(* PLC project Sem nome, Desconhecido Sem nome 1 *)
(* stored: creationDateTime 2019-06-13T18:39:07, modificationDateTime 2019-06-23T17:14:26 *)

PROGRAM program0
  VAR
    saida AT %QX100.0 : BOOL;
    setpoint AT %QW4 : UINT;
    Temperatura AT %IW100 : UINT;
    SaidaAnalog AT %QW100 : UINT;
    Erro AT %QW20 : INT;
    saida2 AT %QX101.0 : BOOL;
    setpoint2 AT %QW8 : UINT;
    Temperatura2 AT %IW102 : UINT;
    SaidaAnalog2 AT %QW101 : UINT;
    Erro2 AT %QW30 : INT;
    aux1 AT %MW200 : UINT;
    aux2 AT %MX202.0 : BOOL;
    aux3 AT %MW204 : UINT;
    aux4 AT %MX202.1 : BOOL;
  END_VAR

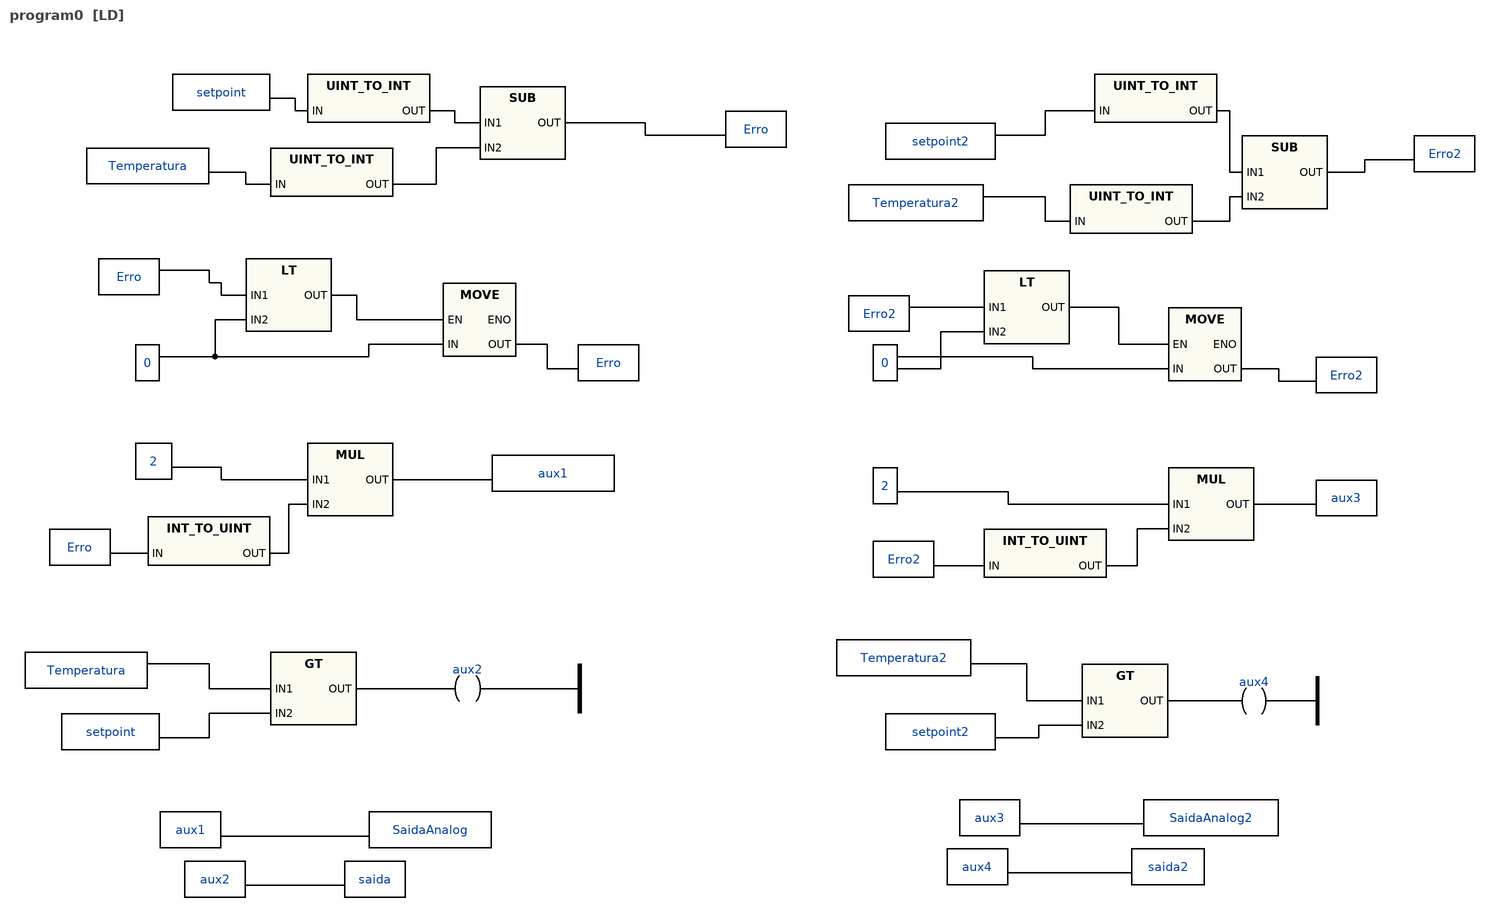
(* LD diagram, written out as Structured Text *)
Erro := UINT_TO_INT(setpoint) - UINT_TO_INT(Temperatura);
Erro2 := UINT_TO_INT(setpoint2) - UINT_TO_INT(Temperatura2);
IF Erro < 0 THEN Erro := 0; END_IF;
IF Erro2 < 0 THEN Erro2 := 0; END_IF;
aux1 := 2 * INT_TO_UINT(Erro);
aux3 := 2 * INT_TO_UINT(Erro2);
aux2 := Temperatura > setpoint;
aux4 := Temperatura2 > setpoint2;
SaidaAnalog2 := aux3;
SaidaAnalog := aux1;
saida2 := aux4;
saida := aux2;
END_PROGRAM

CONFIGURATION Config0
  RESOURCE Res0 ON PLC
    TASK task0(INTERVAL := T#20ms, PRIORITY := 0);
    PROGRAM instance0 WITH task0 : program0;
  END_RESOURCE
END_CONFIGURATION
